PROGRAM decFile
VAR
	s1 : STRING(2000);
	recString: STRING(2047);
	
	fbJson 				: FB_JsonDomParser;
	jsonDoc 			: SJsonValue;
	jsonDoc2 			: SJsonValue;
	jsonProp			: SJsonValue;
	jsonProp2			: SJsonValue;
	jsontempval			: SJsonValue;
	jsontempval2			: SJsonValue;
	jsongettype			: Tc3_JsonXml.EJsonType;
	jsonGetulint		: ULINT;
	jsongetArraySize	: UDINT;
	jsongetArray		: ARRAY[0..1000] OF SJsonValue;
	jsongetArrayulint	: ULINT;
	jsongetArrayudint	: UDINT;
	
	temp 				: STRING;
	btest				: BOOL;
	RisingEdge         : R_TRIG;
	
	JSONVal1 			: STRING;
	JSONVal2 			: STRING;
	
	JSONstr 			: STRING;
	getobj				: INT := 1;
	tempint				: INT;
	
	JSONTEMP			: STRING(2047);
END_VAR

s1 := com.JSONFile;
RisingEdge(CLK:=btest);

IF NOT(s1 = '' AND com.objectread) THEN
	jsonDoc := fbJson.ParseDocument(s1);
	jsonProp :=  fbJson.FindMember(jsonDoc, 'objects');;
	tempint := com.objectNum -1;
	
	IF (jsonProp <> 0) THEN
		jsongettype			:= fbJson.GetType(jsonProp);
		jsongetArraySize	:= fbJson.GetArraySize(jsonProp);
			jsontempval		:= fbJson.GetArrayValueByIdx(jsonProp, (INT_TO_UDINT (tempint) ) );
			JSONTEMP		:= fbJson.GetJson( jsontempval );
				jsonDoc2 			:= fbJson.ParseDocument(JSONTEMP);
				jsonProp2			:= fbJson.FindMember(jsonDoc2, 'centrepointy');
				JSONVal1 			:= fbJson.GetJson(jsonProp2);
				com.objectx			:= STRING_TO_LREAL(JSONVal1);
				
				jsonProp2			:= fbJson.FindMember(jsonDoc2, 'centrepointx');
				JSONVal2 			:= fbJson.GetJson(jsonProp2);
				com.objecty			:= STRING_TO_LREAL(JSONVal2);
	
	END_IF
	
	btest := false;
END_IF

END_PROGRAM

(* stored: Version 1.1.0.1, ProductVersion 3.1.4024.2
   POU decFile: Id {545123ff-5673-497d-8cf4-0c94322715dd}, SpecialFunc None *)
